FUNCTION_BLOCK FB_System
VAR_INPUT
	bStart: BOOL;
	bStop: BOOL;
END_VAR
VAR_OUTPUT
	bInOperation: BOOL;
END_VAR
VAR
	fb_Robot_1: FB_Robot;
	fb_Robot_2: FB_Robot;
	SR_1: SR;
END_VAR

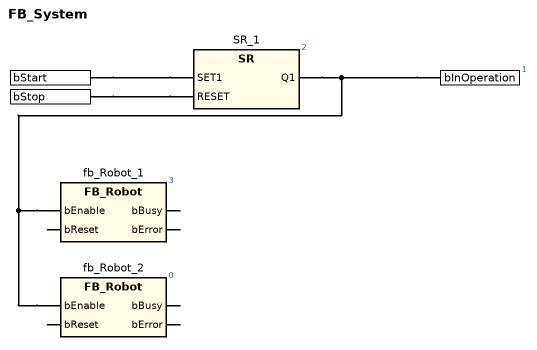
fb_Robot_2(bEnable := SR_1.Q1); // FB_Robot
bInOperation := SR_1.Q1;
SR_1(SET1 := bStart, RESET := bStop); // SR
fb_Robot_1(bEnable := SR_1.Q1); // FB_Robot

END_FUNCTION_BLOCK

(* stored: Version 1.1.0.1, ProductVersion 3.1.4024.11
   POU FB_System: Id {9c58fadf-41db-4240-8a1c-18ce43231fbe}, SpecialFunc None *)
